(* IEC 61131-3 sources: volt/packages/volt-lsp-iec/test-corpus/awa-palletizer/Device/Plc Logic/Application/010 PC01, 8 files *)

(* ---- GLOBAL_CONSTANTS.gvl ---- *)
{attribute 'qualified_only'}
VAR_GLOBAL CONSTANT
END_VAR
VAR_GLOBAL CONSTANT
iProductPositions	: INT := 10;

iSizeRecipesNames 	: INT := 5000;
END_VAR

(* ---- PC01_GVL.gvl ---- *)
{attribute 'qualified_only'}
{attribute 'symbol' := 'none'}
VAR_GLOBAL
	// Button to start the system
	BTN01_Start: libDI;
	// Button to stop the system
	BTN02_Stop: libDI;
	// Button to reset the system
	BTN03_Reset: libDI;
	// Button Emergency Stop
	BTN04_EmergencyStop : libSafetyDI;

	// Unit
	UN01: UN01_Main;

	// Proces Cell
	PC01: PC01_Main;

	// Light On/Off
	SIG01_Red: libSIG;
	// Light On/Off
	SIG02_Orange: libSIG;
	// Light On/Off
	SIG03_Green: libSIG;
	// Light On/Off
	SIG04_Reset: libSIG;
END_VAR

(* ---- PC01_HMI.gvl ---- *)
{attribute 'qualified_only'}
{attribute 'symbol' := 'readwrite'}
VAR_GLOBAL
END_VAR
VAR_GLOBAL
	// Hmi
	{attribute 'symbol' := 'none'}
	BTN01_Start: dutHMI;
	// Hmi
	{attribute 'symbol' := 'none'}
	BTN02_Stop: dutHMI;
	// Hmi
	{attribute 'symbol' := 'none'}
	BTN03_Reset: dutHMI;
	// Hmi
	{attribute 'symbol' := 'none'}
	BTN04_EmergencyStop: dutHMI;

	// Button to start the system
	xBTN01_HmiStart: BOOL := FALSE;
	// Button to stop the system
	xBTN02_HmiStop: BOOL := FALSE;
	// Button to reset the system
	xBTN03_HmiReset: BOOL := FALSE;
	// Button Emergency Stop
	xBTN04_HmiEmergencyStop : BOOL := FALSE;

	// Light On/Off
	SIG01_Red: dutHMI;
	// Light On/Off
	SIG02_Orange: dutHMI;
	// Light On/Off
	SIG03_Green: dutHMI;
	// Light On/Off
	SIG04_Reset: dutHMI;
END_VAR

(* ---- PC01_IO.gvl ---- *)
{attribute 'qualified_only'}
{attribute 'symbol' := 'none'}
VAR_GLOBAL
END_VAR
VAR_GLOBAL
	// Button to start the system
	IxBTN01_Start: BOOL := FALSE;
	// Button to stop the system
	IxBTN02_Stop: BOOL := TRUE;
	// Button to reset the system
	IxBTN03_Reset: BOOL := FALSE;

	IxBTN04_EmergencyStop 	: BOOL := FALSE;		// Button Emergency Stop
	// Light On/Off
	QxSIG01_Red: BOOL := FALSE;
	// Light On/Off
	QxSIG02_Orange: BOOL := FALSE;
	// Light On/Off
	QxSIG03_Green: BOOL := FALSE;
	// Light On/Off
	QxSIG04_Reset: BOOL := FALSE;
END_VAR

(* ---- PC01_PVL.gvl ---- *)
{attribute 'qualified_only'}
VAR_GLOBAL
END_VAR

VAR_GLOBAL RETAIN PERSISTENT
	// Generated instance path of persistent variable
	pgRecipeHandler.RecipeManager.HMI_stRecipeVisu: dutRecipe;
END_VAR
%CLASS PERSISTENT

(* ---- PC01_Safety.gvl ---- *)
{attribute 'qualified_only'}
VAR_GLOBAL
END_VAR

(* ---- PC01_Main.pou ---- *)
FUNCTION_BLOCK PC01_Main
VAR
	// Control module error
	xCMError: BOOL := FALSE;

	//State
	myState : strState;
	// First time init
	xInit: BOOL := TRUE;
	// my handler
	myModuleHandler : L_IMHP_ModuleHandler := (CompType := L_IMHP_ComponentType.GeneralMachineModule);
	ForwardAlarms				: L_IE1P_ForwardSeverity;
	ReadModuleStatus			: L_IE1P_ReadActualSeverity;

	ResetProgramAlarms			: L_IE1P_ResetErrorGlobal;
END_VAR

%LANGUAGE ST
//UNITS - Start/Stop
{region}
	//State control

		IF (xInit) THEN
			xInit := FALSE;
		END_IF

		_Safety();

		PC01_GVL.UN01(IQ_ModuleHandler := myModuleHandler);

	//CONTROL MODULES
	{region}
		PC01_GVL.BTN01_Start(			strName := 'BTN01_Start',
										_HMI := PC01_HMI.BTN01_Start,
										xInput := PC01_IO.IxBTN01_Start OR PC01_HMI.xBTN01_HmiStart,
										tOffDelay := T#100MS,
										tOnDelay  := T#0MS  );

		PC01_GVL.BTN02_Stop(			strName := 'BTN02_Stop',
										_HMI := PC01_HMI.BTN02_Stop,
										xInput := NOT PC01_IO.IxBTN02_Stop OR PC01_HMI.xBTN02_HmiStop,
										tOffDelay := T#100MS,
										tOnDelay  := T#0MS  );

		PC01_GVL.BTN03_Reset(			strName := 'BTN03_Reset',
										_HMI := PC01_HMI.BTN03_Reset,
										xInput := PC01_IO.IxBTN03_Reset OR PC01_HMI.xBTN03_HmiReset,
										tOffDelay := T#100MS,
										tOnDelay  := T#0MS  );

		PC01_GVL.BTN04_EmergencyStop(	strName := 'BTN04_EmergencyStop',
										_HMI := PC01_HMI.BTN04_EmergencyStop,
										xInput := PC01_IO.IxBTN04_EmergencyStop OR PC01_HMI.xBTN04_HmiEmergencyStop,
					  					xCmdReset := PC01_GVL.BTN03_Reset.xDI,
										tOffDelay := T#100MS,
										tOnDelay  := T#0MS  );

		PC01_GVL.SIG01_Red(
							  strName := 'SIG01_Red',
							  _HMI := PC01_HMI.SIG01_Red,
							  xDO       := PC01_GVL.UN01.myState.xStsAborting OR PC01_GVL.UN01.myState.xStsAborted,
							  xDO_Blink := FALSE,
							  xOutput   => PC01_IO.QxSIG01_Red );

		PC01_GVL.SIG02_Orange(
							  strName := 'SIG02_Orange',
							  _HMI := PC01_HMI.SIG02_Orange,
							  xDO       := PC01_GVL.UN01.myState.xStsResetting OR PC01_GVL.UN01.myState.xStsIdle OR
										   PC01_GVL.UN01.myState.xStsStopping OR PC01_GVL.UN01.myState.xStsStopped,
							  xDO_Blink := PC01_GVL.UN01.myState.xStsInit OR PC01_GVL.UN01.myState.xStsResetting,
							  xOutput   => PC01_IO.QxSIG02_Orange);

		PC01_GVL.SIG03_Green(
							  strName := 'SIG03_Green',
							  _HMI := PC01_HMI.SIG03_Green,
							  xDO        := PC01_GVL.UN01.myState.xStsStarting OR PC01_GVL.UN01.myState.xStsExecute,
							  xDO_Blink  := FALSE,
							  xOutput   => PC01_IO.QxSIG03_Green);

		PC01_GVL.SIG04_Reset(
							  strName := 'SIG04_Reset',
							  _HMI := PC01_HMI.SIG04_Reset,
							  xDO	    := TRUE,
					  		  //xDO_Blink := NOT SafetyToPlc.xEmergencyStopOk,
					 		  xOutput   => PC01_IO.QxSIG04_Reset);

		myState.xCmdAbort := PC01_GVL.BTN04_EmergencyStop.xDI OR
							 PC01_GVL.UN01.mystate.xStsAborting OR PC01_GVL.UN01.myState.xStsAborted;
	{endregion}
{endregion}

{region Alarms}
	//------------------------------------------------------------------------------------------------------
	// Alarm and warning handling.
	//------------------------------------------------------------------------------------------------------

	 ReadModuleStatus(xEnable := TRUE,
					ModuleHandler:= myModuleHandler);

	//					OR ReadModuleStatus.eSeverity = L_IE1P_Types.L_IE1P_SeverityLevel.Fault
	//					OR ReadModuleStatus.eSeverity = L_IE1P_Types.L_IE1P_SeverityLevel.Fault_Cinh
	//					OR ReadModuleStatus.eSeverity = L_IE1P_Types.L_IE1P_SeverityLevel.Fault_Log
	//					OR ReadModuleStatus.eSeverity = L_IE1P_Types.L_IE1P_SeverityLevel.Fault_Qsp
	//					OR ReadModuleStatus.eSeverity = L_IE1P_Types.L_IE1P_SeverityLevel.Fault_Qsp_Cinh
	//					OR ReadModuleStatus.eSeverity = L_IE1P_Types.L_IE1P_SeverityLevel.Fault_QspAppl
	//					OR ReadModuleStatus.eReaction >= L_IE1P_Types.L_IE1P_Reaction.NormalStop;
	//					OR ReadModuleStatus.eSeverity = L_IE1P_Types.L_IE1P_SeverityLevel.Warning
	//					OR ReadModuleStatus.eSeverity = L_IE1P_Types.L_IE1P_SeverityLevel.Warning_Lock;

	 ForwardAlarms(
		xEnable:= TRUE,
		ModuleHandler:= myModuleHandler,
		xForwardFromChildModules:=TRUE);
{endregion}

END_FUNCTION_BLOCK

ACTION _Safety
%LANGUAGE ST
//
// Safety communication.
//

END_ACTION

(* ---- pgPC01.pou ---- *)
PROGRAM pgPC01
VAR
END_VAR

%LANGUAGE ST
PC01_GVL.PC01();

END_PROGRAM
